FUNCTION_BLOCK Counter
  (* Version 0.1, 2005-12-27, Oscar Ljungkrantz, Chalmers *)
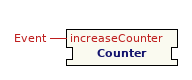
  EVENT_INPUT
    increaseCounter;
  END_EVENT
  VAR
    value : INT := 0;
    streng : WSTRING := litetesttext;
  END_VAR
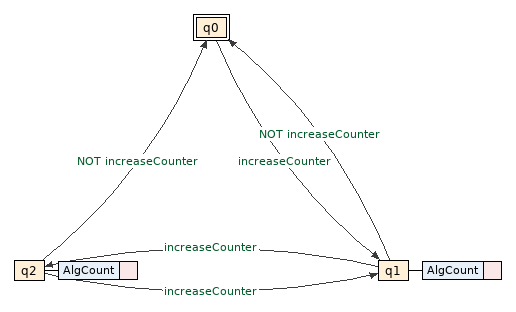
  EC_STATES
    q0;
    q1 : AlgCount;
    q2 : AlgCount;
  END_STATES
  EC_TRANSITIONS
    q0 TO q1 := increaseCounter;
    q1 TO q2 := increaseCounter;
    q1 TO q0 := NOT increaseCounter;
    q2 TO q1 := increaseCounter;
    q2 TO q0 := NOT increaseCounter;
  END_TRANSITIONS
  ALGORITHM AlgCount IN Java:
		value++;
		System.out.println("Value: " + value);
  END_ALGORITHM
END_FUNCTION_BLOCK
(* other elements stored in the file *)
(* Algorithm Name="AlgCount" Comment="Normally executed algorithm" > <ST Text="System.out.println();" /> </Algorithm *)
